// TIA Portal V18 program export: 1 tag tables, 0 data types, 0 data blocks, 2 code blocks (in call order from the OBs), 0 instance data blocks

VAR_GLOBAL   // PLC tag table "Default tag table"
   Start AT %M0.0 : Bool;
   Fan AT %Q0.0 : Bool;
   "Fan Out Delay" AT %MD2 : Time;
   "Element Start" AT %M0.1 : Bool;
   Element AT %Q0.2 : Bool;
   "Element Time Delay" AT %MD6 : Time;
   "Start Up" AT %M0.2 : Bool;
   "Start Up Delay" AT %MD10 : Time;
   Auger AT %Q0.1 : Bool;
   RTD AT %IW96 : Word;
   "RTD 2" AT %IW98 : Word;
   Setpoint AT %MW20 : Word;
   "RTD Real" AT %MD14 : Real;
   "RTD 2 Real" AT %MD22 : Real;
   "Corrected RTD Temp" AT %MD26 : Real;
   "Corrected RTD 2 Temp" AT %MD30 : Real;
   "Auger PID" AT %M0.3 : Bool;
   "Corrected Setpoint" AT %MD34 : Real;
   "Auger Start Up" AT %M0.4 : Bool;
   "Auger Duty Cycle Start" AT %M0.5 : Bool;
   "Auger Duty Cycle" AT %M0.6 : Bool;
   "Auger Duty Cycle Output" AT %M0.7 : Bool;
   "Test Output" AT %M1.0 : Bool;
   "Set Reset" AT %M1.1 : Bool;
   "Error Ack" AT %M1.2 : Bool;
   "Error Ack Button" AT %M1.3 : Bool;
END_VAR

ORGANIZATION_BLOCK "Main"   // OB1, LAD, ProgramCycle
TITLE = "Main Program Sweep (Cycle)"
{ S7_Optimized_Access := 'TRUE' }
VERSION : 0.1
// stored: AutoNumber true, IsIECCheckEnabled false, SetENOAutomatically false
   VAR_INPUT
      Initial_Call : Bool;   // Initial call of this OB
      Remanence : Bool;   // =True, if remanent data are available
   END_VAR
   VAR_TEMP   // added for the SCL form of the ladder/FBD networks
      _w1 : Bool;
   END_VAR
BEGIN

REGION Network 1
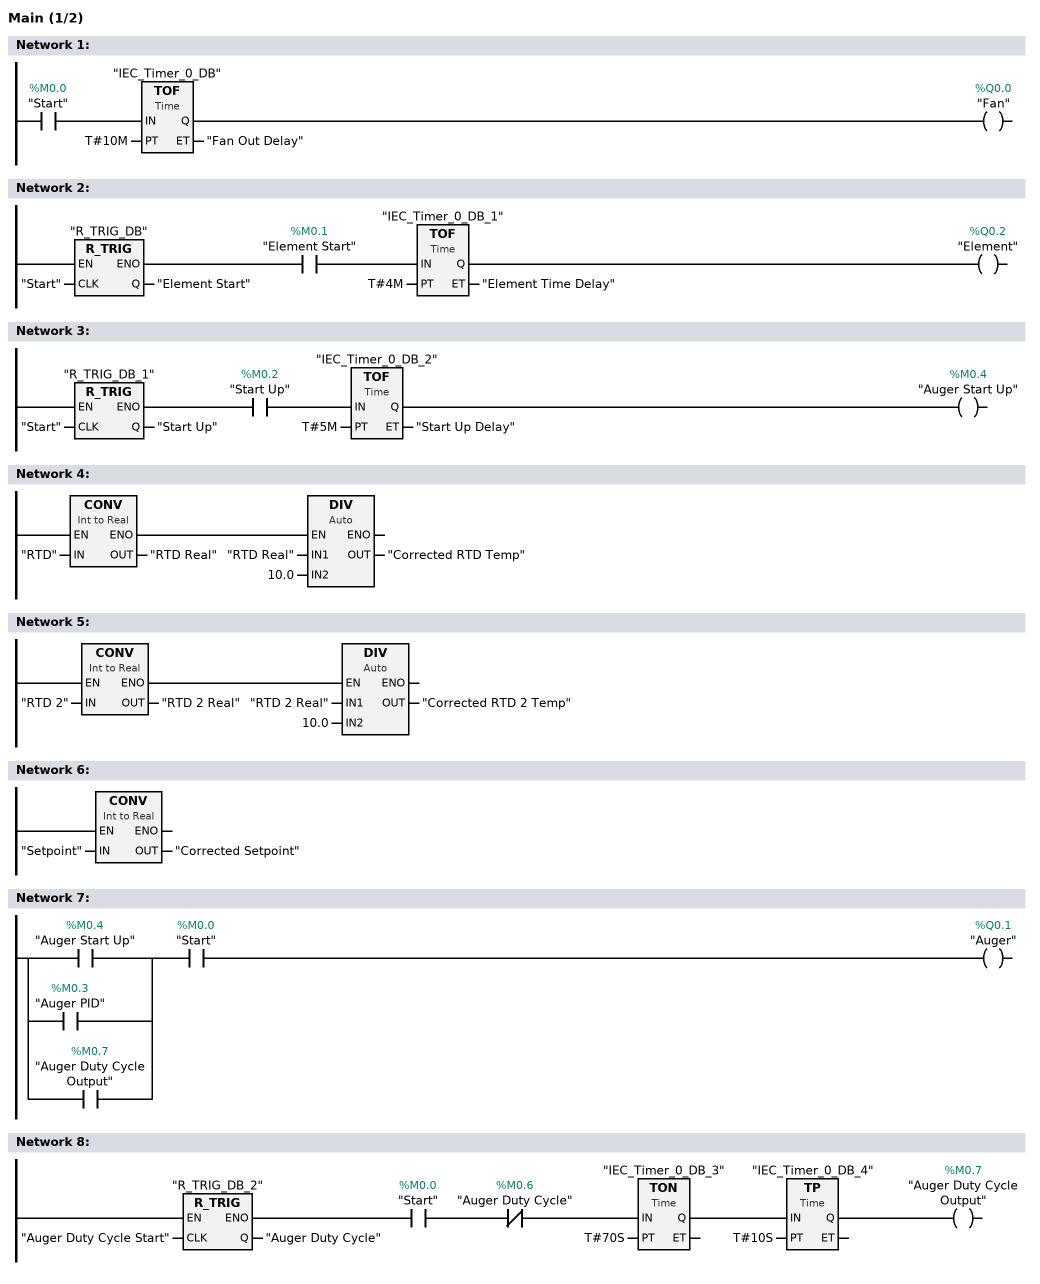
   RUNG wire#powerrail
      Contact( "Start" )
      { S7_Templates := "time_type := Time" } "IEC_Timer_0_DB".TOF(pt := T#10M, et => "Fan Out Delay")
      Coil( "Fan" )
   END_RUNG
   // the same network as SCL:
   "IEC_Timer_0_DB".TOF(IN := "Start", PT := T#10M, ET => "Fan Out Delay");
   "Fan" := "IEC_Timer_0_DB".Q;
END_REGION

REGION Network 2
   RUNG wire#powerrail
      "R_TRIG_DB".R_TRIG(CLK := "Start", Q => "Element Start")
      Contact( "Element Start" )
      { S7_Templates := "time_type := Time" } "IEC_Timer_0_DB_1".TOF(pt := T#4M, et => "Element Time Delay")
      Coil( "Element" )
   END_RUNG
   // the same network as SCL:
   "R_TRIG_DB"(CLK := "Start", Q => "Element Start", ENO => #_w1);   // R_TRIG
   "IEC_Timer_0_DB_1".TOF(IN := #_w1 AND "Element Start", PT := T#4M, ET => "Element Time Delay");
   "Element" := "IEC_Timer_0_DB_1".Q;
END_REGION

REGION Network 3
   RUNG wire#powerrail
      "R_TRIG_DB_1".R_TRIG(CLK := "Start", Q => "Start Up")
      Contact( "Start Up" )
      { S7_Templates := "time_type := Time" } "IEC_Timer_0_DB_2".TOF(pt := T#5M, et => "Start Up Delay")
      Coil( "Auger Start Up" )
   END_RUNG
   // the same network as SCL:
   "R_TRIG_DB_1"(CLK := "Start", Q => "Start Up", ENO => #_w1);   // R_TRIG
   "IEC_Timer_0_DB_2".TOF(IN := #_w1 AND "Start Up", PT := T#5M, ET => "Start Up Delay");
   "Auger Start Up" := "IEC_Timer_0_DB_2".Q;
END_REGION

REGION Network 4
   RUNG wire#powerrail
      { S7_Templates := "[SrcType := Int, DestType := Real]" } Convert(in := "RTD", out => "RTD Real")
      Div(in1 := "RTD Real", in2 := 10.0, out => "Corrected RTD Temp")
   END_RUNG
   // the same network as SCL:
   "RTD Real" := INT_TO_REAL("RTD");
   "Corrected RTD Temp" := "RTD Real" / 10.0;
END_REGION

REGION Network 5
   RUNG wire#powerrail
      { S7_Templates := "[SrcType := Int, DestType := Real]" } Convert(in := "RTD 2", out => "RTD 2 Real")
      Div(in1 := "RTD 2 Real", in2 := 10.0, out => "Corrected RTD 2 Temp")
   END_RUNG
   // the same network as SCL:
   "RTD 2 Real" := INT_TO_REAL("RTD 2");
   "Corrected RTD 2 Temp" := "RTD 2 Real" / 10.0;
END_REGION

REGION Network 6
   RUNG wire#powerrail
      { S7_Templates := "[SrcType := Int, DestType := Real]" } Convert(in := "Setpoint", out => "Corrected Setpoint")
   END_RUNG
   // the same network as SCL:
   "Corrected Setpoint" := INT_TO_REAL("Setpoint");
END_REGION

REGION Network 7
   RUNG wire#powerrail
      Contact( "Auger Start Up" )
      wire#w1
      Contact( "Start" )
      Coil( "Auger" )
   END_RUNG
   RUNG wire#powerrail
      Contact( "Auger PID" )
   END_RUNG wire#w1
   RUNG wire#powerrail
      Contact( "Auger Duty Cycle Output" )
   END_RUNG wire#w1
   // the same network as SCL:
   "Auger" := ("Auger Start Up" OR "Auger PID" OR "Auger Duty Cycle Output") AND "Start";
END_REGION

REGION Network 8
   RUNG wire#powerrail
      "R_TRIG_DB_2".R_TRIG(CLK := "Auger Duty Cycle Start", Q => "Auger Duty Cycle")
      Contact( "Start" )
      I_Contact( "Auger Duty Cycle" )
      { S7_Templates := "time_type := Time" } "IEC_Timer_0_DB_3".TON(pt := T#70S, et =>)
      { S7_Templates := "time_type := Time" } "IEC_Timer_0_DB_4".TP(pt := T#10S, et =>)
      Coil( "Auger Duty Cycle Output" )
   END_RUNG
   // the same network as SCL:
   "R_TRIG_DB_2"(CLK := "Auger Duty Cycle Start", Q => "Auger Duty Cycle", ENO => #_w1);   // R_TRIG
   "IEC_Timer_0_DB_3".TON(IN := #_w1 AND "Start" AND NOT "Auger Duty Cycle", PT := T#70S);
   "IEC_Timer_0_DB_4".TP(IN := "IEC_Timer_0_DB_3".Q, PT := T#10S);
   "Auger Duty Cycle Output" := "IEC_Timer_0_DB_4".Q;
END_REGION

REGION Network 9
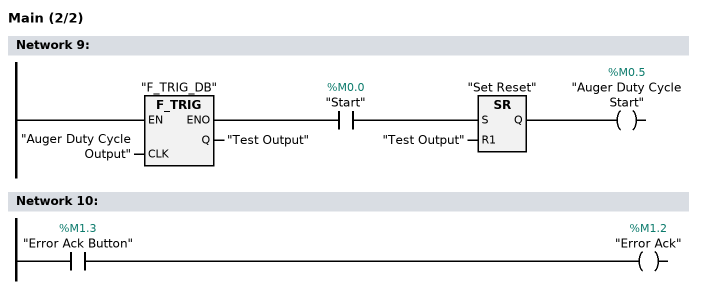
   RUNG wire#powerrail
      "F_TRIG_DB".F_TRIG(CLK := "Auger Duty Cycle Output", Q => "Test Output")
      Contact( "Start" )
      S_SR(operand := "Set Reset", r1 := "Test Output")
      Coil( "Auger Duty Cycle Start" )
   END_RUNG
   // the same network as SCL:
   "F_TRIG_DB"(CLK := "Auger Duty Cycle Output", Q => "Test Output", ENO => #_w1);   // F_TRIG
   IF #_w1 AND "Start" THEN
       "Set Reset" := TRUE;   // SR flip-flop
   END_IF;
   IF "Test Output" THEN "Set Reset" := FALSE; END_IF;
   "Auger Duty Cycle Start" := "Set Reset";
END_REGION

REGION Network 10
   RUNG wire#powerrail
      Contact( "Error Ack Button" )
      Coil( "Error Ack" )
   END_RUNG
   // the same network as SCL:
   "Error Ack" := "Error Ack Button";
END_REGION
END_ORGANIZATION_BLOCK

ORGANIZATION_BLOCK "Cyclic interrupt"   // OB30, LAD, CyclicInterrupt
{ S7_Optimized_Access := 'TRUE' }
VERSION : 0.1
// stored: AutoNumber true, IsIECCheckEnabled false, SetENOAutomatically false
   VAR_INPUT
      Initial_Call : Bool;   // Initial call of this OB
      Event_Count : Int;   // Events discarded
   END_VAR
BEGIN

REGION Network 1
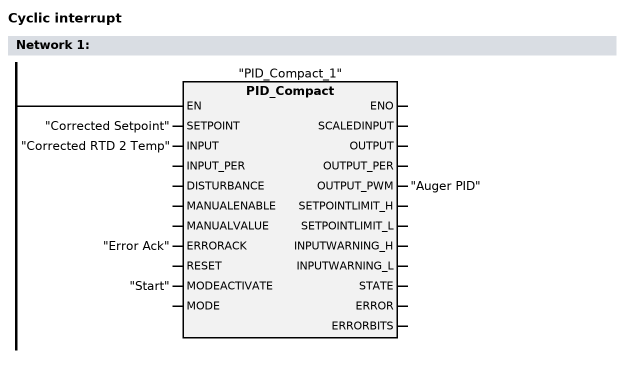
   RUNG wire#powerrail
      "PID_Compact_1".PID_Compact(Setpoint := "Corrected Setpoint", Input := "Corrected RTD 2 Temp", Input_PER :=, Disturbance :=, ManualEnable :=, ManualValue :=, ErrorAck := "Error Ack", Reset :=, ModeActivate := "Start", Mode :=, ScaledInput =>, Output =>, Output_PER =>, Output_PWM => "Auger PID", SetpointLimit_H =>, SetpointLimit_L =>, InputWarning_H =>, InputWarning_L =>, State =>, Error =>, ErrorBits =>)
   END_RUNG
   // the same network as SCL:
   "PID_Compact_1"(Setpoint := "Corrected Setpoint",   // PID_Compact
                   Input := "Corrected RTD 2 Temp",
                   ErrorAck := "Error Ack",
                   ModeActivate := "Start",
                   Output_PWM => "Auger PID");
END_REGION
END_ORGANIZATION_BLOCK
